TYPE TFPortaManCmd :
STRUCT
	ApriPorta : BOOL;
	ChiudiPorta : bool;
END_STRUCT
END_TYPE

(* stored: Version 1.1.0.1, ProductVersion 3.1.4024.11
   DUT TFPortaManCmd: Id {884f6cce-8377-46c9-ac4a-b317a8e1e314} *)
